// TIA Portal V15.1 export
// export: Created 2020-06-12T07:35:53.3974609Z, ExportSetting None, DisplayName Totally Integrated Automation Portal, DisplayVersion V15.1, DisplayName TIA Portal Openness, DisplayVersion V15.1, DisplayName STEP 7 Professional, DisplayVersion V15.1, DisplayName STEP 7 Safety, DisplayVersion V15.1, DisplayName WinCC Advanced, DisplayVersion V15.1
FUNCTION "L15_Recipe" : Void   // FC99, FBD
{ S7_Optimized_Access := 'TRUE' }
// stored: SetENOAutomatically False
   VAR_TEMP
      par375 : Bool;
      par460 : Bool;
      par504 : Bool;
      par540 : Bool;
      par594 : Bool;
      par750 : Bool;
      tMoldFlowMax : Real;
      tMoldFlowMin : Real;
      tBaseFlowMax : Real;
      tBaseFlowMin : Real;
      tBand1 : Real;
      tBand2 : Real;
      tBand3 : Real;
      tBand4 : Real;
      tBand5 : Real;
      tBand6 : Real;
      tBand7 : Real;
      tElecDiaR : DInt;
      tElecDia : Real;
      tParamID : Int;
      tEleID : Int;
      tVarI1 : Int;
      tStartTime : Real;
      tIdx : Int;
      tStartAmount : Real;
      tFeedingTime : Real;
      tApply : Bool;
      tApplyForMS1 : Bool;
      tApplyForMS2 : Bool;
      tGasPressMelt : Real;
      tGasPressHT : Real;
      tGasPressNorm : Real;
      tMoldDia : Real;
      tLength : Real;
      tVolume : Real;
      tUpdate : Bool;
      tReadBack : Bool;
      tEnaStore : Bool;
      tDisStore : Bool;
      tCheckFixSTT : Bool;
      tCheckFixHTT : Bool;
      tDummy : Bool;
      tCopyFromBackup : Bool;
   END_VAR
   VAR_TEMP   // added for the SCL form of the ladder/FBD networks
      _w1 : Bool;
      _w2 : Bool;
      _w3 : Bool;
      _w4 : Bool;
   END_VAR
BEGIN

REGION Network 1: Calculate the electrode ID
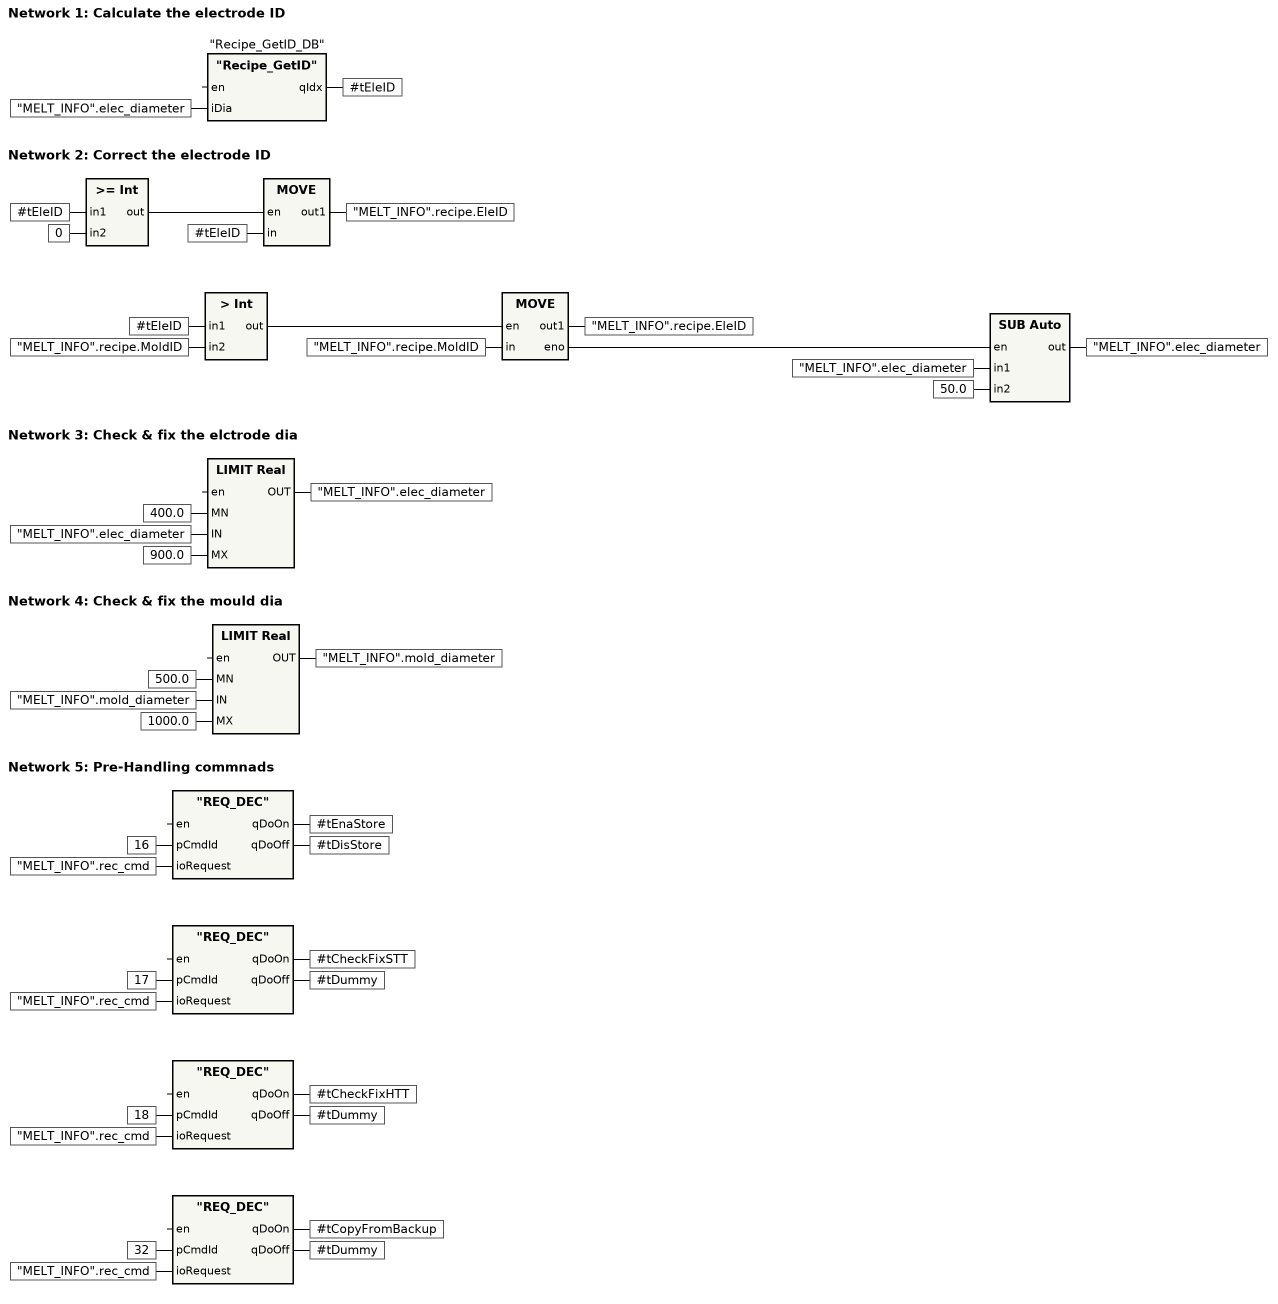
   "Recipe_GetID_DB"(iDia := "MELT_INFO".elec_diameter, qIdx => #tEleID);   // "Recipe_GetID"
END_REGION

REGION Network 2: Correct the electrode ID
   IF #tEleID >= 0 THEN "MELT_INFO".recipe.EleID := #tEleID; END_IF;
   IF #tEleID > "MELT_INFO".recipe.MoldID THEN
       "MELT_INFO".recipe.EleID := "MELT_INFO".recipe.MoldID;
       "MELT_INFO".elec_diameter := "MELT_INFO".elec_diameter - 50.0;
   END_IF;
END_REGION

REGION Network 3: Check & fix the elctrode dia
   "MELT_INFO".elec_diameter := LIMIT(MN := 400.0, IN := "MELT_INFO".elec_diameter, MX := 900.0);
END_REGION

REGION Network 4: Check & fix the mould dia
   "MELT_INFO".mold_diameter := LIMIT(MN := 500.0, IN := "MELT_INFO".mold_diameter, MX := 1000.0);
END_REGION

REGION Network 5: Pre-Handling commnads
   "REQ_DEC"(pCmdId := 16, ioRequest := "MELT_INFO".rec_cmd, qDoOn => #tEnaStore, qDoOff => #tDisStore);
   "REQ_DEC"(pCmdId := 17, ioRequest := "MELT_INFO".rec_cmd, qDoOn => #tCheckFixSTT, qDoOff => #tDummy);
   "REQ_DEC"(pCmdId := 18, ioRequest := "MELT_INFO".rec_cmd, qDoOn => #tCheckFixHTT, qDoOff => #tDummy);
   "REQ_DEC"(pCmdId := 32, ioRequest := "MELT_INFO".rec_cmd, qDoOn => #tCopyFromBackup, qDoOff => #tDummy);
END_REGION

REGION Network 6: Database entries editing
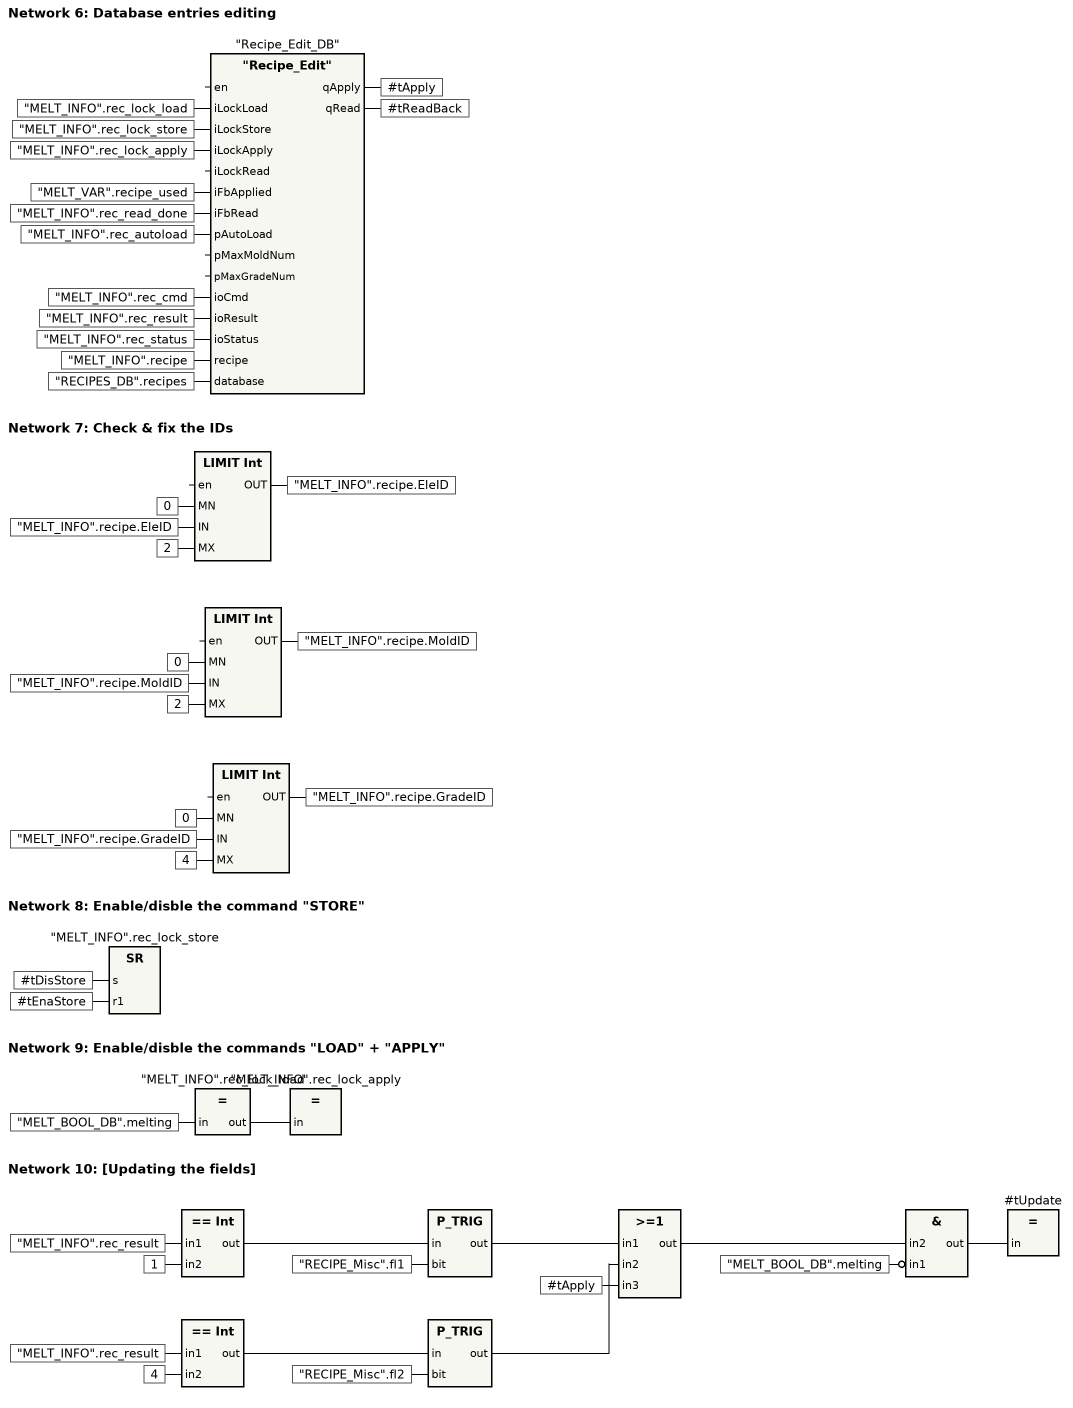
   "Recipe_Edit_DB"(iLockLoad := "MELT_INFO".rec_lock_load,   // "Recipe_Edit"
                    iLockStore := "MELT_INFO".rec_lock_store,
                    iLockApply := "MELT_INFO".rec_lock_apply,
                    iFbApplied := "MELT_VAR".recipe_used,
                    iFbRead := "MELT_INFO".rec_read_done,
                    pAutoLoad := "MELT_INFO".rec_autoload,
                    ioCmd := "MELT_INFO".rec_cmd,
                    ioResult := "MELT_INFO".rec_result,
                    ioStatus := "MELT_INFO".rec_status,
                    recipe := "MELT_INFO".recipe,
                    database := "RECIPES_DB".recipes,
                    qApply => #tApply,
                    qRead => #tReadBack);
END_REGION

REGION Network 7: Check & fix the IDs
   "MELT_INFO".recipe.EleID := LIMIT(MN := 0, IN := "MELT_INFO".recipe.EleID, MX := 2);
   "MELT_INFO".recipe.MoldID := LIMIT(MN := 0, IN := "MELT_INFO".recipe.MoldID, MX := 2);
   "MELT_INFO".recipe.GradeID := LIMIT(MN := 0, IN := "MELT_INFO".recipe.GradeID, MX := 4);
END_REGION

REGION Network 8: Enable/disble the command "STORE"
   IF #tDisStore THEN
       "MELT_INFO".rec_lock_store := TRUE;   // SR flip-flop
   END_IF;
   IF #tEnaStore THEN "MELT_INFO".rec_lock_store := FALSE; END_IF;
END_REGION

REGION Network 9: Enable/disble the commands "LOAD" + "APPLY"
   "MELT_INFO".rec_lock_load := "MELT_BOOL_DB".melting;
   "MELT_INFO".rec_lock_apply := "MELT_BOOL_DB".melting;
END_REGION

REGION Network 10: [Updating the fields]
   #_w1 := "MELT_INFO".rec_result = 1;
   #_w2 := #_w1 AND NOT "RECIPE_Misc".fl1;   // rising edge
   "RECIPE_Misc".fl1 := #_w1;
   #_w3 := "MELT_INFO".rec_result = 4;
   #_w4 := #_w3 AND NOT "RECIPE_Misc".fl2;   // rising edge
   "RECIPE_Misc".fl2 := #_w3;
   #tUpdate := (#_w2 OR #_w4 OR #tApply) AND NOT "MELT_BOOL_DB".melting;
END_REGION

REGION Network 11 (SCL): The field to update during recipe editing
   IF #tUpdate THEN
       "MELT_INFO".mold_diameter := INT_TO_REAL("MELT_INFO".mold_geo["MELT_INFO".recipe.MoldID].dia);
       "MELT_INFO".mold_length := INT_TO_REAL("MELT_INFO".mold_geo["MELT_INFO".recipe.MoldID].length);
       //
       "MELT_VAR".calc_el_wht := "MELT_INFO".elec_weight;
       "MELT_VAR".calc_stub_wht := "MELT_INFO".stub_weight;
       "MELT_INFO".steel_density := "MELT_INFO".recipe.steel_density;
   END_IF;
   #tMoldDia := "MELT_INFO".mold_diameter * "MELT_INFO".recipe.ingot_shrink_factor / 1000.0;
   #tLength := "MELT_INFO".mold_length / 1000.0;
   #tVolume := 3.14159 * #tLength * #tMoldDia ** 2 / 4;
   // beacuse there is slag inside the maximum weight must be reduced
   // to simplify the calculation we use factor 0.9
   "MELT_INFO".ingot_weight_max := 0.9 * #tVolume * ("MELT_INFO".steel_density * 1000.0);
END_REGION

REGION Network 12 (SCL): Use the same timetable for the P and R curves
   IF #tCheckFixSTT THEN
       "MELT_INFO".recipe.ST_R.x := "MELT_INFO".recipe.ST_P.x;
   ELSIF #tCheckFixHTT THEN
       "MELT_INFO".recipe.HT_R.x := "MELT_INFO".recipe.HT_P.x;
   END_IF;
END_REGION

REGION Network 13: [[ APPLY / COPY TO ]]
END_REGION

REGION Network 14: [ Cooling parameters ]
END_REGION

REGION Network 15: CW parameters: dT
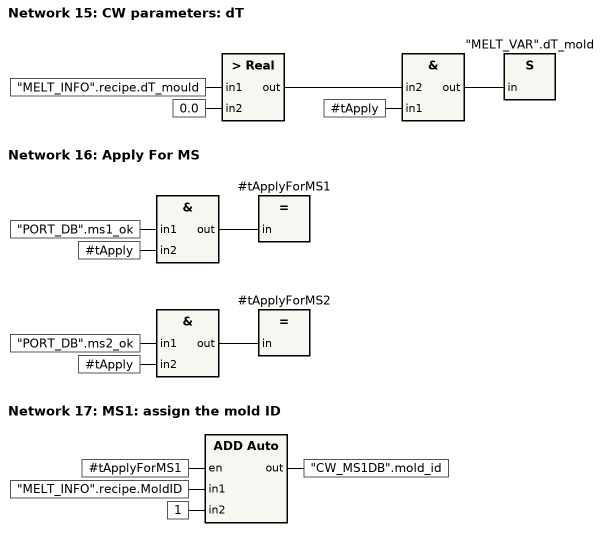
   IF ("MELT_INFO".recipe.dT_mould > 0.0) AND #tApply THEN "MELT_VAR".dT_mold := TRUE; END_IF;
END_REGION

REGION Network 16: Apply For MS
   #tApplyForMS1 := "PORT_DB".ms1_ok AND #tApply;
   #tApplyForMS2 := "PORT_DB".ms2_ok AND #tApply;
END_REGION

REGION Network 17: MS1: assign the mold ID
   IF #tApplyForMS1 THEN "CW_MS1DB".mold_id := "MELT_INFO".recipe.MoldID + 1; END_IF;
END_REGION

REGION Network 18: MS1: cooling parameters
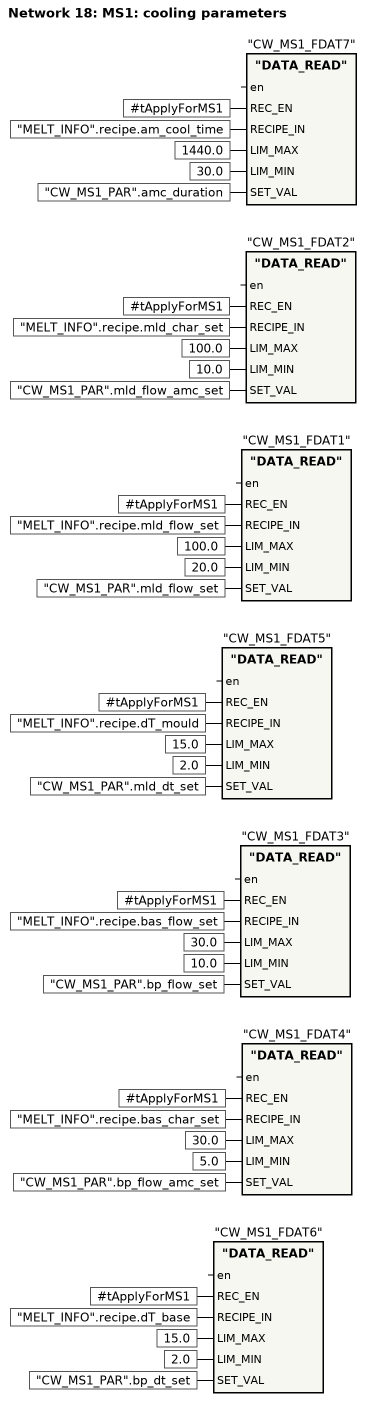
   "CW_MS1_FDAT7"(REC_EN := #tApplyForMS1,   // "DATA_READ"
                  RECIPE_IN := "MELT_INFO".recipe.am_cool_time,
                  LIM_MAX := 1440.0,
                  LIM_MIN := 30.0,
                  SET_VAL := "CW_MS1_PAR".amc_duration);
   "CW_MS1_FDAT2"(REC_EN := #tApplyForMS1,   // "DATA_READ"
                  RECIPE_IN := "MELT_INFO".recipe.mld_char_set,
                  LIM_MAX := 100.0,
                  LIM_MIN := 10.0,
                  SET_VAL := "CW_MS1_PAR".mld_flow_amc_set);
   "CW_MS1_FDAT1"(REC_EN := #tApplyForMS1,   // "DATA_READ"
                  RECIPE_IN := "MELT_INFO".recipe.mld_flow_set,
                  LIM_MAX := 100.0,
                  LIM_MIN := 20.0,
                  SET_VAL := "CW_MS1_PAR".mld_flow_set);
   "CW_MS1_FDAT5"(REC_EN := #tApplyForMS1,   // "DATA_READ"
                  RECIPE_IN := "MELT_INFO".recipe.dT_mould,
                  LIM_MAX := 15.0,
                  LIM_MIN := 2.0,
                  SET_VAL := "CW_MS1_PAR".mld_dt_set);
   "CW_MS1_FDAT3"(REC_EN := #tApplyForMS1,   // "DATA_READ"
                  RECIPE_IN := "MELT_INFO".recipe.bas_flow_set,
                  LIM_MAX := 30.0,
                  LIM_MIN := 10.0,
                  SET_VAL := "CW_MS1_PAR".bp_flow_set);
   "CW_MS1_FDAT4"(REC_EN := #tApplyForMS1,   // "DATA_READ"
                  RECIPE_IN := "MELT_INFO".recipe.bas_char_set,
                  LIM_MAX := 30.0,
                  LIM_MIN := 5.0,
                  SET_VAL := "CW_MS1_PAR".bp_flow_amc_set);
   "CW_MS1_FDAT6"(REC_EN := #tApplyForMS1,   // "DATA_READ"
                  RECIPE_IN := "MELT_INFO".recipe.dT_base,
                  LIM_MAX := 15.0,
                  LIM_MIN := 2.0,
                  SET_VAL := "CW_MS1_PAR".bp_dt_set);
END_REGION

REGION Network 19: MS2: assign the mold ID
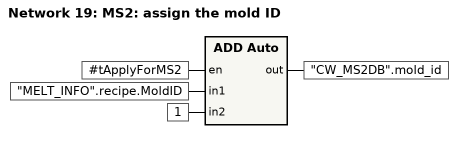
   IF #tApplyForMS2 THEN "CW_MS2DB".mold_id := "MELT_INFO".recipe.MoldID + 1; END_IF;
END_REGION

REGION Network 20: MS2: cooling parameters
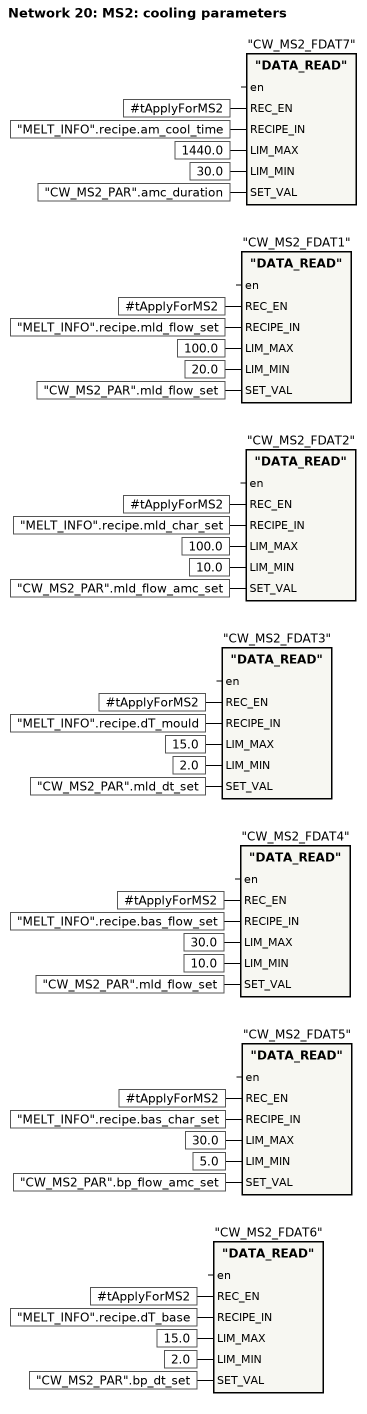
   "CW_MS2_FDAT7"(REC_EN := #tApplyForMS2,   // "DATA_READ"
                  RECIPE_IN := "MELT_INFO".recipe.am_cool_time,
                  LIM_MAX := 1440.0,
                  LIM_MIN := 30.0,
                  SET_VAL := "CW_MS2_PAR".amc_duration);
   "CW_MS2_FDAT1"(REC_EN := #tApplyForMS2,   // "DATA_READ"
                  RECIPE_IN := "MELT_INFO".recipe.mld_flow_set,
                  LIM_MAX := 100.0,
                  LIM_MIN := 20.0,
                  SET_VAL := "CW_MS2_PAR".mld_flow_set);
   "CW_MS2_FDAT2"(REC_EN := #tApplyForMS2,   // "DATA_READ"
                  RECIPE_IN := "MELT_INFO".recipe.mld_char_set,
                  LIM_MAX := 100.0,
                  LIM_MIN := 10.0,
                  SET_VAL := "CW_MS2_PAR".mld_flow_amc_set);
   "CW_MS2_FDAT3"(REC_EN := #tApplyForMS2,   // "DATA_READ"
                  RECIPE_IN := "MELT_INFO".recipe.dT_mould,
                  LIM_MAX := 15.0,
                  LIM_MIN := 2.0,
                  SET_VAL := "CW_MS2_PAR".mld_dt_set);
   "CW_MS2_FDAT4"(REC_EN := #tApplyForMS2,   // "DATA_READ"
                  RECIPE_IN := "MELT_INFO".recipe.bas_flow_set,
                  LIM_MAX := 30.0,
                  LIM_MIN := 10.0,
                  SET_VAL := "CW_MS2_PAR".mld_flow_set);
   "CW_MS2_FDAT5"(REC_EN := #tApplyForMS2,   // "DATA_READ"
                  RECIPE_IN := "MELT_INFO".recipe.bas_char_set,
                  LIM_MAX := 30.0,
                  LIM_MIN := 5.0,
                  SET_VAL := "CW_MS2_PAR".bp_flow_amc_set);
   "CW_MS2_FDAT6"(REC_EN := #tApplyForMS2,   // "DATA_READ"
                  RECIPE_IN := "MELT_INFO".recipe.dT_base,
                  LIM_MAX := 15.0,
                  LIM_MIN := 2.0,
                  SET_VAL := "CW_MS2_PAR".bp_dt_set);
END_REGION

REGION Network 21: [Process parameters]
END_REGION

REGION Network 22 (SCL): Curves
   IF #tApply THEN
       "MELT_VAR".ST_P := "MELT_INFO".recipe.ST_P;
       "MELT_VAR".ST_R := "MELT_INFO".recipe.ST_R;
       "MELT_VAR".HT_P := "MELT_INFO".recipe.HT_P;
       "MELT_VAR".HT_R := "MELT_INFO".recipe.HT_R;
   END_IF;
END_REGION

REGION Network 23 (SCL): Speed controller parameters
   IF #tApply THEN
       "MELT_CONT_EL_ID".PSET1 := "MELT_INFO".recipe.vxc_param1;
       "MELT_CONT_EL_ID".PSET2 := "MELT_INFO".recipe.vxc_param2;
   END_IF;
END_REGION

REGION Network 24 (SCL): Melt controllers parameters
   IF #tApply THEN
       // meltrate controller
       "MELT_VAR".use_mr := "MELT_INFO".recipe.mode_mt_mr;
       "MELT_CONT_DB".mr_set := "MELT_INFO".recipe.meltrate;
       "MELT_CONT_MR_ID".pSET := "MELT_INFO".recipe.mrc_param;
       // swing controllers
       "MELT_VAR".use_sw := "MELT_INFO".recipe.mode_mt_sw;
       "MELT_VAR".swc_on_st_delay := "MELT_INFO".recipe.sw_del;
       "MELT_CONT_DB".sw_set := "MELT_INFO".recipe.swing;
       "MELT_CONT_SW_ID".pSET := "MELT_INFO".recipe.swc_param;
   END_IF;
END_REGION

REGION Network 25: Hottoping start/stop parameters
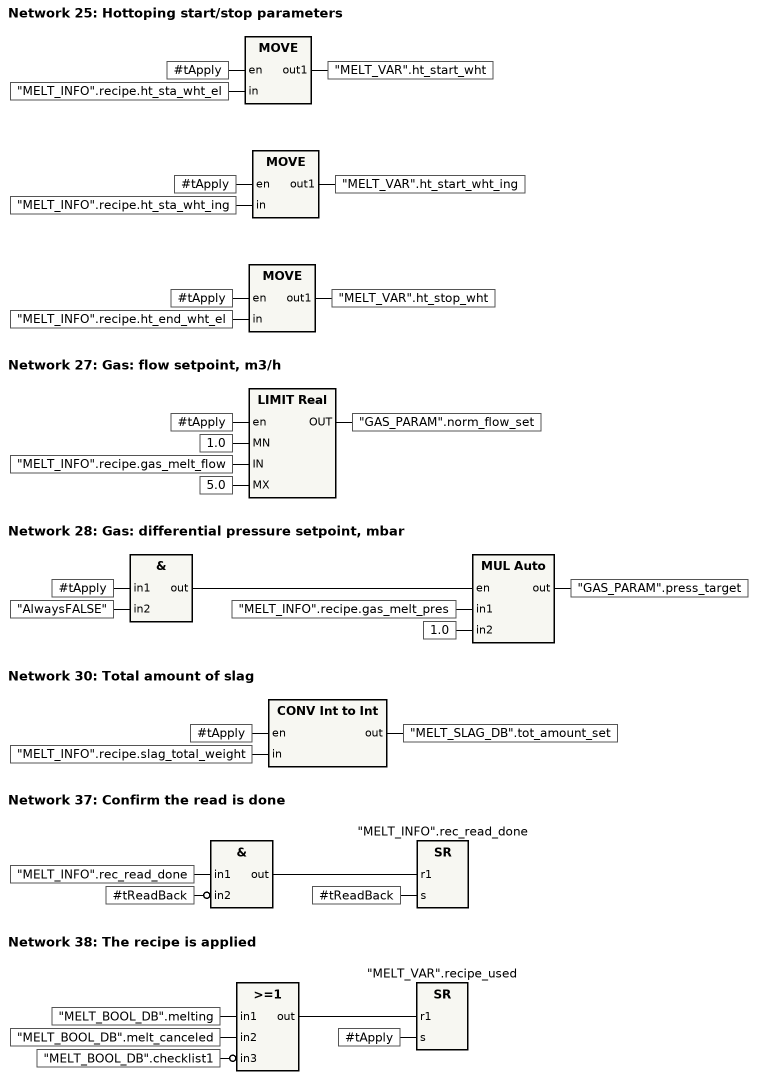
   IF #tApply THEN
       "MELT_VAR".ht_start_wht := "MELT_INFO".recipe.ht_sta_wht_el;
       "MELT_VAR".ht_start_wht_ing := "MELT_INFO".recipe.ht_sta_wht_ing;
       "MELT_VAR".ht_stop_wht := "MELT_INFO".recipe.ht_end_wht_el;
   END_IF;
END_REGION

REGION Network 26: [Gas]
END_REGION

REGION Network 27: Gas: flow setpoint, m3/h
   IF #tApply THEN
       "GAS_PARAM".norm_flow_set := LIMIT(MN := 1.0, IN := "MELT_INFO".recipe.gas_melt_flow, MX := 5.0);
   END_IF;
END_REGION

REGION Network 28: Gas: differential pressure setpoint, mbar
   // The diff.pressure setpoint is useless for this plant
   IF #tApply AND "AlwaysFALSE" THEN
       "GAS_PARAM".press_target := "MELT_INFO".recipe.gas_melt_pres * 1.0;
   END_IF;
END_REGION

REGION Network 29: [Slag parameters]
END_REGION

REGION Network 30: Total amount of slag
   IF #tApply THEN "MELT_SLAG_DB".tot_amount_set := INT_TO_INT("MELT_INFO".recipe.slag_total_weight); END_IF;
END_REGION

REGION Network 31 (SCL): Prepare weight setpoints (start slag, base slag, feeding rate)
   IF #tApply THEN
       //start slag parameters calculation
       "MELT_SLAG_DB".tot_amount_set := "MELT_INFO".recipe.slag_total_weight;
       #tStartAmount :=
       INT_TO_REAL("MELT_INFO".recipe.slag_start_weight)
       * INT_TO_REAL("MELT_SLAG_DB".tot_amount_set) / 100.0;
       "MELT_SLAG_DB".start_amount_set := ROUND_INT(#tStartAmount);
       // base slag parameters calculation
       #tStartTime := 0;
       FOR #tIdx := 1 TO 8 DO
           IF #tStartTime < "MELT_INFO".recipe.ST_P.x[#tIdx] THEN
               #tStartTime := "MELT_INFO".recipe.ST_P.x[#tIdx];
           END_IF;
       END_FOR;
       IF #tStartTime < 5 THEN
           #tStartTime := 30;
       END_IF;
       // cacluate duration
       #tFeedingTime := INT_TO_REAL("MELT_INFO".recipe.slag_duration) / 100.0;
       IF #tFeedingTime <= 0.0 OR #tFeedingTime >= 0.95 THEN
           #tFeedingTime := 0.5; 
       END_IF;
       "MELT_SLAG_DB".base_load_delay := "MELT_INFO".recipe.slag_delay;
       "MELT_SLAG_DB".base_load_time_set := #tStartTime * #tFeedingTime;
       "MELT_SLAG_DB".base_slag_rate := INT_TO_REAL("MELT_SLAG_DB".base_amount_set) / "MELT_SLAG_DB".base_load_time_set;
   END_IF;
END_REGION

REGION Network 32: [[ READ BACK / COPY FROM ]]
END_REGION

REGION Network 33 (SCL): Curves
   IF #tReadBack THEN
       "MELT_INFO".recipe.ST_P := "MELT_VAR".ST_P;
       "MELT_INFO".recipe.ST_R := "MELT_VAR".ST_R;
       "MELT_INFO".recipe.HT_P := "MELT_VAR".HT_P;
       "MELT_INFO".recipe.HT_R := "MELT_VAR".HT_R;
   END_IF;
END_REGION

REGION Network 34 (SCL): Speed controller parameters
   IF #tReadBack THEN
       "MELT_INFO".recipe.vxc_param1 := "MELT_CONT_EL_ID".PSET1;
       "MELT_INFO".recipe.vxc_param2 := "MELT_CONT_EL_ID".PSET2;
   END_IF;
END_REGION

REGION Network 35 (SCL): MR/SW controllers parameters
   IF #tReadBack THEN
       // meltrate controller
       "MELT_INFO".recipe.meltrate := "MELT_CONT_DB".mr_set;
       "MELT_INFO".recipe.mrc_param := "MELT_CONT_MR_ID".pSET;
       // swing controllers
       "MELT_INFO".recipe.swing := "MELT_CONT_DB".sw_set;
       "MELT_INFO".recipe.swc_param := "MELT_CONT_SW_ID".pSET;
   END_IF;
END_REGION

REGION Network 36 (SCL): Slag addition parameters
   IF #tReadBack THEN
       "MELT_INFO".recipe.slag_total_weight := "MELT_SLAG_DB".tot_amount_set;
       "MELT_INFO".recipe.slag_start_weight := ROUND_INT("MELT_SLAG_DB".start_amount_set / "MELT_SLAG_DB".tot_amount_set * 100.0);
       "MELT_INFO".recipe.slag_delay := ROUND_INT("MELT_SLAG_DB".base_load_delay);
       // find the duration of the starting phase
       #tStartTime := 0;
       FOR #tIdx := 1 TO 8 DO
           IF #tStartTime < "MELT_INFO".recipe.ST_P.x[#tIdx] THEN
               #tStartTime := "MELT_INFO".recipe.ST_P.x[#tIdx];
           END_IF;
       END_FOR;
       "MELT_INFO".recipe.slag_duration := ROUND_INT("MELT_SLAG_DB".base_load_time_set / #tStartTime * 100.0);
   END_IF;
END_REGION

REGION Network 37: Confirm the read is done
   #_w1 := "MELT_INFO".rec_read_done AND NOT #tReadBack;
   IF #tReadBack THEN
       "MELT_INFO".rec_read_done := TRUE;   // SR flip-flop
   END_IF;
   IF #_w1 THEN "MELT_INFO".rec_read_done := FALSE; END_IF;
END_REGION

REGION Network 38: The recipe is applied
   IF #tApply THEN
       "MELT_VAR".recipe_used := TRUE;   // SR flip-flop
   END_IF;
   IF "MELT_BOOL_DB".melting OR "MELT_BOOL_DB".melt_canceled OR NOT "MELT_BOOL_DB".checklist1 THEN
       "MELT_VAR".recipe_used := FALSE;
   END_IF;
END_REGION

REGION Network 39 (SCL): Copy from BACKUP
   IF #tCopyFromBackup THEN
       FOR #tIdx := 0 TO 60 DO
           "RECIPES_DB".recipes[#tIdx] := "RECIPES_BU_DB".THIS[#tIdx];
       END_FOR;
   END_IF;
END_REGION

REGION Network 40: [[END]]
END_REGION
END_FUNCTION
